// TIA Portal V19 export
TYPE "LAF_typeDevDiagState"
TITLE = PN device diag state bit coded / PN device diag Status bitcodiert
// This data type contains the status information of the devices and represents a user interface. / PN device Diagnose
// stored: Access Published
   STRUCT
      configured { ExternalAccessible := 'False'; ExternalVisible := 'False'; ExternalWritable := 'False'} : Bool;   // konfiguriert - mittels "DeviceStates" / Configured, identified by "DeviceStates"
      faulty { ExternalAccessible := 'False'; ExternalVisible := 'False'; ExternalWritable := 'False'} : Bool;   // gestört - mittels "DeviceStates" / Faulty, identified by "DeviceStates"
      deactivated { ExternalAccessible := 'False'; ExternalVisible := 'False'; ExternalWritable := 'False'} : Bool;   // deaktiviert - mittels "DeviceStates" / Dectivated, identified by "DeviceStates"
      present { ExternalAccessible := 'False'; ExternalVisible := 'False'; ExternalWritable := 'False'} : Bool;   // vorhanden - mittels "DeviceStates" / Existing, identified by "DeviceStates"
      problem { ExternalAccessible := 'False'; ExternalVisible := 'False'; ExternalWritable := 'False'} : Bool;   // Problem - mittels "DeviceStates" !!! welche Probleme gibt es, und wie sind diese genauer zu spezifizieren !!! / Problem identified by "DeviceStates"
      networkError { ExternalAccessible := 'False'; ExternalVisible := 'False'; ExternalWritable := 'False'} : Bool;   // Netzwerk-Fehler / Network error
      maintenanceRequired { ExternalAccessible := 'False'; ExternalVisible := 'False'; ExternalWritable := 'False'} : Bool;   // Maintenance Required / Wartungsbedarf
      maintenanceDemanded { ExternalAccessible := 'False'; ExternalVisible := 'False'; ExternalWritable := 'False'} : Bool;   // Maintenance Demanded / Wartungsanforderung
      wasFaulty { ExternalAccessible := 'False'; ExternalVisible := 'False'; ExternalWritable := 'False'} : Bool;   // War gestört; gebildet aus Faulty (speichernd) - mittels "DeviceStates" / Was faulty, identified by "DeviceStates"
      wasProblem { ExternalAccessible := 'False'; ExternalVisible := 'False'; ExternalWritable := 'False'} : Bool;   // War Problem; gebildet aus Problem (speichernd) - mittels "DeviceStates" / There was a problem, identified by "DeviceStates"
      modulStateSummary { ExternalAccessible := 'False'; ExternalVisible := 'False'; ExternalWritable := 'False'} : Bool;   // Summenstatus aller unterlagerten Module - mittels Bit0 "ModuleStates" / Summary modul state identified by "ModuleStates", Bit0
      spare11 { ExternalAccessible := 'False'; ExternalVisible := 'False'; ExternalWritable := 'False'} : Bool;   // Reserve / Spare
      spare12 { ExternalAccessible := 'False'; ExternalVisible := 'False'; ExternalWritable := 'False'} : Bool;   // Reserve / Spare
      spare13 { ExternalAccessible := 'False'; ExternalVisible := 'False'; ExternalWritable := 'False'} : Bool;   // Reserve / Spare
      spare14 { ExternalAccessible := 'False'; ExternalVisible := 'False'; ExternalWritable := 'False'} : Bool;   // Reserve / Spare
      spare15 { ExternalAccessible := 'False'; ExternalVisible := 'False'; ExternalWritable := 'False'} : Bool;   // Reserve / Spare
   END_STRUCT;
END_TYPE
